//==================================================================================================
//							Beckhoff Automation Poland
//									18.04.2018
//	Struktura zawierajaca I/O odpowiedniego bloku
//  v1.0	|| TC v 3.1.4022.16		|| - pierwsza wersja
//==================================================================================================
TYPE ST_MCReadParameterSetIO :
STRUCT
	bExecute						: BOOL;								// Rising edge executes cmd
	bDone							: BOOL;
	bBusy							: BOOL;
	bError							: BOOL;
	udiErrorID						: UDINT;
END_STRUCT
END_TYPE

(* stored: Version 1.1.0.1, ProductVersion 3.1.4022.12
   DUT ST_MCReadParameterSetIO: Id {12f30249-5fc1-4095-82be-2e45a3a6b0e5} *)
